TYPE UDT_VacuumAdmin :
STRUCT
	i: UDT_VacuumInput;
	o: UDT_VacuumOutput;
END_STRUCT
END_TYPE

(* stored: Version 1.1.0.1, ProductVersion 3.1.4022.16
   DUT UDT_VacuumAdmin: Id {5042d5f5-c6aa-48fb-8777-9743491251f3} *)
